// TIA Portal V19 export
TYPE "HU_Pump_Par"
// stored: Access Published
   STRUCT
      DelayCheckFilterClogged : Time := T#1M;
      DelayPumpInactivity : Time := T#15M;
      DelayEvPressureStart : Time := T#500MS;
      DelayEvPressureStop : Time := T#1M;
      DelayPressureRunning : Time;
   END_STRUCT;
END_TYPE
